% RSLogix 500 project I2P HANDS-ON 3 - ANDREW.RSS, saved by version 10.00.00.00 %
PROJECT "UNTITLED"    % processor: Bul.1763 MicroLogix 1100 Series B %

PROGRAM FILES
  LAD 2   10 rungs

DATA FILES
  O0 OUTPUT  4 elements
  I1 INPUT  6 elements
  S2 STATUS  66 elements
  B3 BINARY  1 elements
  T4 TIMER  1 elements
  C5 COUNTER  1 elements
  R6 CONTROL  1 elements
  N7 INTEGER  1 elements
  F8 FLOAT  1 elements

LADDER 2
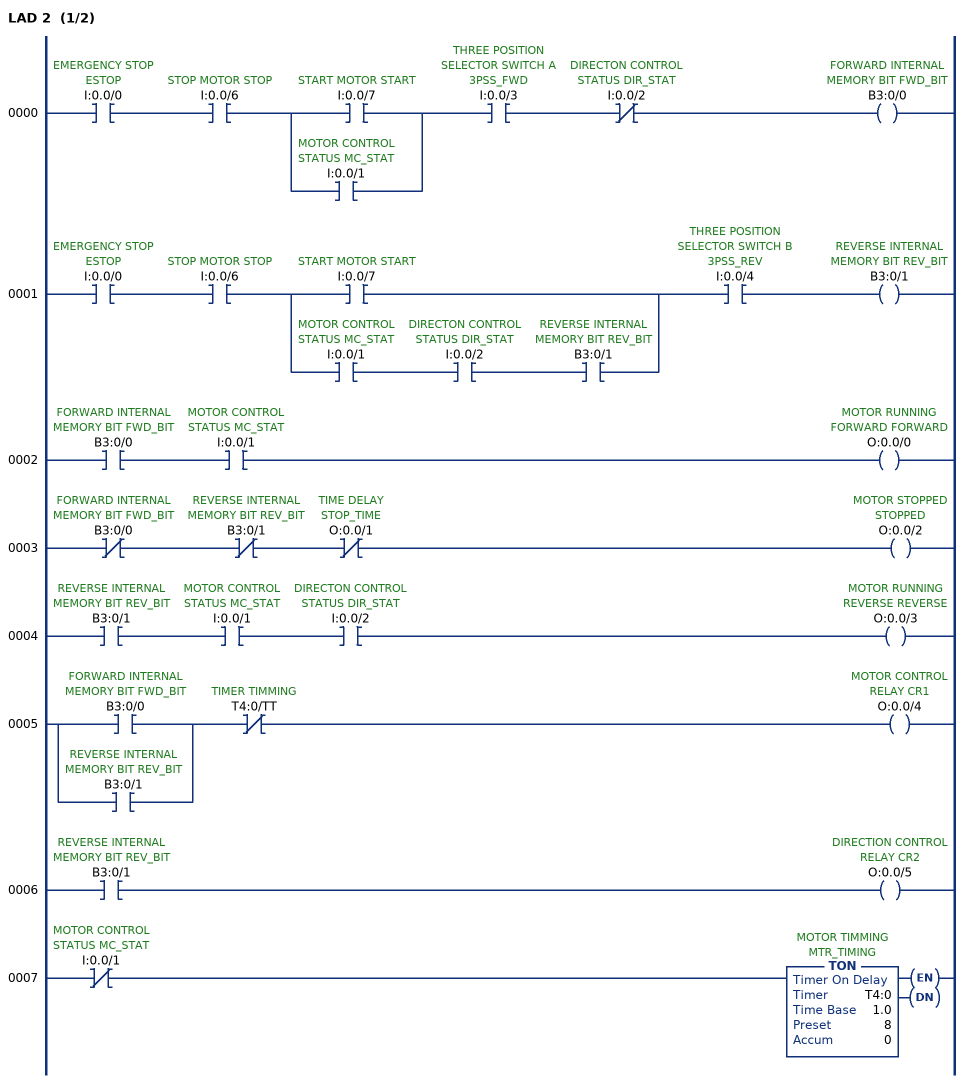
% Rung: 0 %
SOR XIC I:0.0/0 XIC I:0.0/6 BST XIC I:0.0/7 NXB XIC I:0.0/1 BND XIC I:0.0/3 XIO I:0.0/2 OTE B3:0/0 EOR
%   I:0.0/0  ESTOP  "EMERGENCY STOP" %
%   I:0.0/6  STOP  "STOP MOTOR" %
%   I:0.0/7  START  "START MOTOR" %
%   I:0.0/1  MC_STAT  "MOTOR CONTROL STATUS" %
%   I:0.0/3  3PSS_FWD  "THREE POSITION SELECTOR SWITCH A" %
%   I:0.0/2  DIR_STAT  "DIRECTON CONTROL STATUS" %
%   B3:0/0  FWD_BIT  "FORWARD INTERNAL MEMORY BIT" %
% Rung: 1 %
SOR XIC I:0.0/0 XIC I:0.0/6 BST XIC I:0.0/7 NXB XIC I:0.0/1 XIC I:0.0/2 XIC B3:0/1 BND XIC I:0.0/4 OTE B3:0/1 EOR
%   I:0.0/0  ESTOP  "EMERGENCY STOP" %
%   I:0.0/6  STOP  "STOP MOTOR" %
%   I:0.0/7  START  "START MOTOR" %
%   I:0.0/1  MC_STAT  "MOTOR CONTROL STATUS" %
%   I:0.0/2  DIR_STAT  "DIRECTON CONTROL STATUS" %
%   B3:0/1  REV_BIT  "REVERSE INTERNAL MEMORY BIT" %
%   I:0.0/4  3PSS_REV  "THREE POSITION SELECTOR SWITCH B" %
% Rung: 2 %
SOR XIC B3:0/0 XIC I:0.0/1 OTE O:0.0/0 EOR
%   B3:0/0  FWD_BIT  "FORWARD INTERNAL MEMORY BIT" %
%   I:0.0/1  MC_STAT  "MOTOR CONTROL STATUS" %
%   O:0.0/0  FORWARD  "MOTOR RUNNING FORWARD" %
% Rung: 3 %
SOR XIO B3:0/0 XIO B3:0/1 XIO O:0.0/1 OTE O:0.0/2 EOR
%   B3:0/0  FWD_BIT  "FORWARD INTERNAL MEMORY BIT" %
%   B3:0/1  REV_BIT  "REVERSE INTERNAL MEMORY BIT" %
%   O:0.0/1  STOP_TIME  "TIME DELAY" %
%   O:0.0/2  STOPPED  "MOTOR STOPPED" %
% Rung: 4 %
SOR XIC B3:0/1 XIC I:0.0/1 XIC I:0.0/2 OTE O:0.0/3 EOR
%   B3:0/1  REV_BIT  "REVERSE INTERNAL MEMORY BIT" %
%   I:0.0/1  MC_STAT  "MOTOR CONTROL STATUS" %
%   I:0.0/2  DIR_STAT  "DIRECTON CONTROL STATUS" %
%   O:0.0/3  REVERSE  "MOTOR RUNNING REVERSE" %
% Rung: 5 %
SOR BST XIC B3:0/0 NXB XIC B3:0/1 BND XIO T4:0/TT OTE O:0.0/4 EOR
%   B3:0/0  FWD_BIT  "FORWARD INTERNAL MEMORY BIT" %
%   B3:0/1  REV_BIT  "REVERSE INTERNAL MEMORY BIT" %
%   T4:0/TT  "TIMER TIMMING" %
%   O:0.0/4  CR1  "MOTOR CONTROL RELAY" %
% Rung: 6 %
SOR XIC B3:0/1 OTE O:0.0/5 EOR
%   B3:0/1  REV_BIT  "REVERSE INTERNAL MEMORY BIT" %
%   O:0.0/5  CR2  "DIRECTION CONTROL RELAY" %
% Rung: 7 %
SOR XIO I:0.0/1 TON T4:0 1.0 8 0 EOR
%   I:0.0/1  MC_STAT  "MOTOR CONTROL STATUS" %
%   T4:0  MTR_TIMING  "MOTOR TIMMING" %

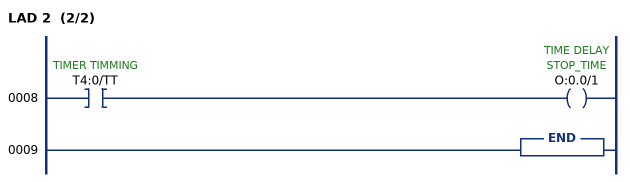
% Rung: 8 %
SOR XIC T4:0/TT OTE O:0.0/1 EOR
%   T4:0/TT  "TIMER TIMMING" %
%   O:0.0/1  STOP_TIME  "TIME DELAY" %
% Rung: 9 %
SOR END EOR

OTHER DOCUMENTED ADDRESSES
  I:0.0/5  2PSS  "TWO POSITION SLECTOR SWITCH"
  I:0.0/8  PB3_NO  "PUSHBUTTON 3 NO"

DATA TABLE (non-zero values as saved)
DATA T4
% .PRE .ACC %
% T4:0 % 8 0
